TYPE ST_GC_Admin :
STRUCT
	bLocalControl : BOOL;
END_STRUCT
END_TYPE

(* stored: Version 1.1.0.1, ProductVersion 3.1.4026.18
   DUT ST_GC_Admin: Id {9d771c70-165f-48ed-a888-a145a70861d4} *)
